// TIA Portal V19 export
TYPE "_IOL_VM_TPV70_10"
   STRUCT
      StandardStructure : Struct   // Tetra Pak V70 DeviceID:10
         Header : Struct
            NumberParameter : Int := 4;   // Number of device parameters (Device Identification + Device Parameter)
            AdressParamDownLoad : Int := 20;   // Start adress for ParamDownload signals in this struct
            AdressDeviceIndent : Int;   // Start adress for Device Identification Parameters in this struct (82 Bytes ea)
            AdressApplicSpez : Int;   // Start adress ApplicationSpezificTag (82 Bytes ea) [9]
            AdressDeviceParam : Int := 44;   // Start adress for Device Parameters in this Area (20 Bytes ea) [15]
            AdressKommando : Int;   // Start adress for Device Commandos
            NumberCommandos : Int;   // Number of Commandos of the device
            Spare01 : Int;   // spare
            Spare02 : Int;   // spare
            Spare03 : Int;   // spare
         END_STRUCT;
         Paramdownload : Struct
            ParamDownLoadStart : Struct   // Parameter Download Start (Only if master and device are V1.1)
               BlockStat : DWord;   // function block status
               IOLStat : DWord;   // IO-Link Status
            END_STRUCT;
            ParamDownLoadEnd : Struct   // Parameter Download End (Only if master and device are V1.1)
               BlockStat : DWord;   // function block status
               IOLStat : DWord;   // IO-Link Status
            END_STRUCT;
            ParamDownLoadStore : Struct   // Parameter Download Store (Only if master and device are V1.1)
               BlockStat : DWord;   // function block status
               IOLStat : DWord;   // IO-Link Status
            END_STRUCT;
         END_STRUCT;
         Parameter : Struct   // Address Device Indent
            SV1Avtivations : Struct
               value : DInt;
            END_STRUCT;
            Index : Int := 83;   // parameter index
            Subindex : Int := 1;   // parameter subindex
            Length : Int := 4;   // parameter length in BYTE for writing
            BlockStat : DWord;   // function block status
            IOLStat : DWord;   // IO-Link Status
            RelRead : Bool := TRUE;   // reading release
            RelWrite : Bool;   // writing release
         END_STRUCT;
         Parameter1 : Struct   // Address Device Indent
            SV1_EnDuration : Struct
               value : DInt;
            END_STRUCT;
            Index : Int := 85;   // parameter index
            Subindex : Int := 1;   // parameter subindex
            Length : Int := 4;   // parameter length in BYTE for writing
            BlockStat : DWord;   // function block status
            IOLStat : DWord;   // IO-Link Status
            RelRead : Bool := TRUE;   // reading release
            RelWrite : Bool;   // writing release
         END_STRUCT;
         Parameter2 : Struct   // Address Device Indent
            SV1_DeEnDuration : Struct
               value : DInt;
            END_STRUCT;
            Index : Int := 86;   // parameter index
            Subindex : Int := 1;   // parameter subindex
            Length : Int := 4;   // parameter length in BYTE for writing
            BlockStat : DWord;   // function block status
            IOLStat : DWord;   // IO-Link Status
            RelRead : Bool := TRUE;   // reading release
            RelWrite : Bool;   // writing release
         END_STRUCT;
         Parameter3 : Struct   // Address Device Indent
            ObjErrorTime : Struct
               value : Byte;
               spacer : Array[0..1] of Byte;
            END_STRUCT;
            Index : Int := 70;   // parameter index
            Subindex : Int := 1;   // parameter subindex
            Length : Int := 1;   // parameter length in BYTE for writing
            BlockStat : DWord;   // function block status
            IOLStat : DWord;   // IO-Link Status
            RelRead : Bool := TRUE;   // reading release
            RelWrite : Bool;   // writing release
         END_STRUCT;
      END_STRUCT;
   END_STRUCT;
END_TYPE
